# EPICS substitutions: db/Beckhoff_5XXX/ecmcEL5101-0011.substitutions
file "ecmcEcSlave.template"
{
  pattern {}
          {}
}

file "ecmcEL5101-0011-chX.template"
{
  pattern { CH_ID, DTYP,             FTVL }
          { 01,    asynInt32ArrayIn, LONG }
}
